FUNCTION_BLOCK LOADLE (* LOADL with QI Enable *)
  (* Standard: 61499-2; Classification: Simulation *)
  (* Version 0.0, 2004-11-08, JHC, Rockwell Automation, Derived from LOADL. *)
  (* Compiler header: package fb.rt.mva; import fb.rt.net.*; *)
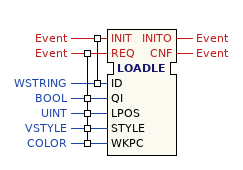
  EVENT_INPUT
    INIT WITH ID; (* Service Initialization *)
    REQ WITH LPOS, STYLE, WKPC, QI; (* Publish LOAD command *)
  END_EVENT
  EVENT_OUTPUT
    INITO; (* Initialization Confirm *)
    CNF; (* Execution Confirmation *)
  END_EVENT
  VAR_INPUT
    ID : WSTRING; (* Local Group ID, default = FB instance name *)
    QI : BOOL; (* 0=Disable, 1=Enable *)
    LPOS : UINT; (* Load Position in % of Conveyor Length *)
    STYLE : VSTYLE := NONE; (* Input Workpiece style *)
    WKPC : COLOR := yellow; (* Input Workpiece Color *)
  END_VAR
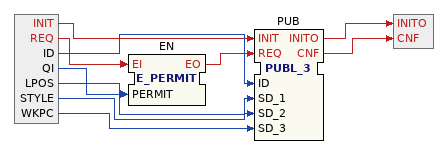
  FBS
    PUB : PUBL_3;
    EN : E_PERMIT;
  END_FBS
  EVENT_CONNECTIONS
    INIT TO PUB.INIT;
    PUB.INITO TO INITO;
    PUB.CNF TO CNF;
    REQ TO EN.EI;
    EN.EO TO PUB.REQ;
  END_CONNECTIONS
  DATA_CONNECTIONS
    ID TO PUB.ID;
    LPOS TO PUB.SD_1;
    STYLE TO PUB.SD_2;
    WKPC TO PUB.SD_3;
    QI TO EN.PERMIT;
  END_CONNECTIONS
END_FUNCTION_BLOCK
